TYPE (* AUX Output Color and Picture *)
  (* Description: Copyright (c) 2025 HR Agrartechnik GmbH This program and the accompanying materials are made available under the terms of the Eclipse Public License 2.0 which is available at https://www.eclipse.org/legal/epl-2.0/ SPDX-License-Identifier: EPL-2.0 *)
  (* Version 1.0, 2025-06-12, Franz Höpfinger, HR Agrartechnik GmbH *)
  PACKAGE logiBUS::utils::sequence::schieber;
  IMPORT isobus::ut::IDs::ID_NULL;
  IMPORT isobus::ut::colours::COLOR_WHITE;
  SchieberAuxOutStruct : STRUCT
    Picture : UINT := ID_NULL; (* u16ObjId for Picture *)
    u8Colour : USINT := COLOR_WHITE; (* Background Color of the AUX *)
  END_STRUCT;
END_TYPE
